{attribute 'qualified_only'}
{attribute 'strict'}
TYPE E_ROOM_TEMP_STS :
(
	baixa:=1,
	normal:=2,
	moderada:=3,
	alta:=4,
	muito_alta:=5
);
END_TYPE

(* stored: Version 1.1.0.1, ProductVersion 3.1.4024.11
   DUT E_ROOM_TEMP_STS: Id {9242d6f2-7607-4296-b47c-673b40174353} *)
